INTERFACE ITcoControlVoltage

PROPERTY IsOff : BOOL
GET
END_GET
END_PROPERTY

PROPERTY IsOn : BOOL
GET
END_GET
END_PROPERTY

END_INTERFACE

(* stored: Version 1.1.0.1
   Itf ITcoControlVoltage: Id {37533fcd-a138-4914-8d22-78d3f1e02647}
   Property IsOff: Id {e5e14c33-cc81-420f-9d61-8e40d8609390}
   Get Get: Id {5d08b90e-aa45-4ab0-a9b3-c602cc73cf1b}
   Property IsOn: Id {b2a27d1b-2ace-4b88-be87-f0483bcb3c8e}
   Get Get: Id {bd391189-747a-4f0d-b358-940e49182478} *)
